PROGRAM C05_MachineStatus
VAR
	fbMachinState					: FB_SYSTEM_MachineState;

	fbPowerDelay					: TOF;
	tofEUCAPassthroughDisableDelay	: TOF;
	ftrigPassthroughCheck			: F_TRIG;
	ftrigConditionalRunOff			: F_TRIG;

	tonPowerUpTimer				: TON;
	tonEUCAMachineRun			: TON;

END_VAR
VAR // added by the converter: edge detectors and wires of the graphical bodies
    _w1, _w2 : BOOL;
END_VAR

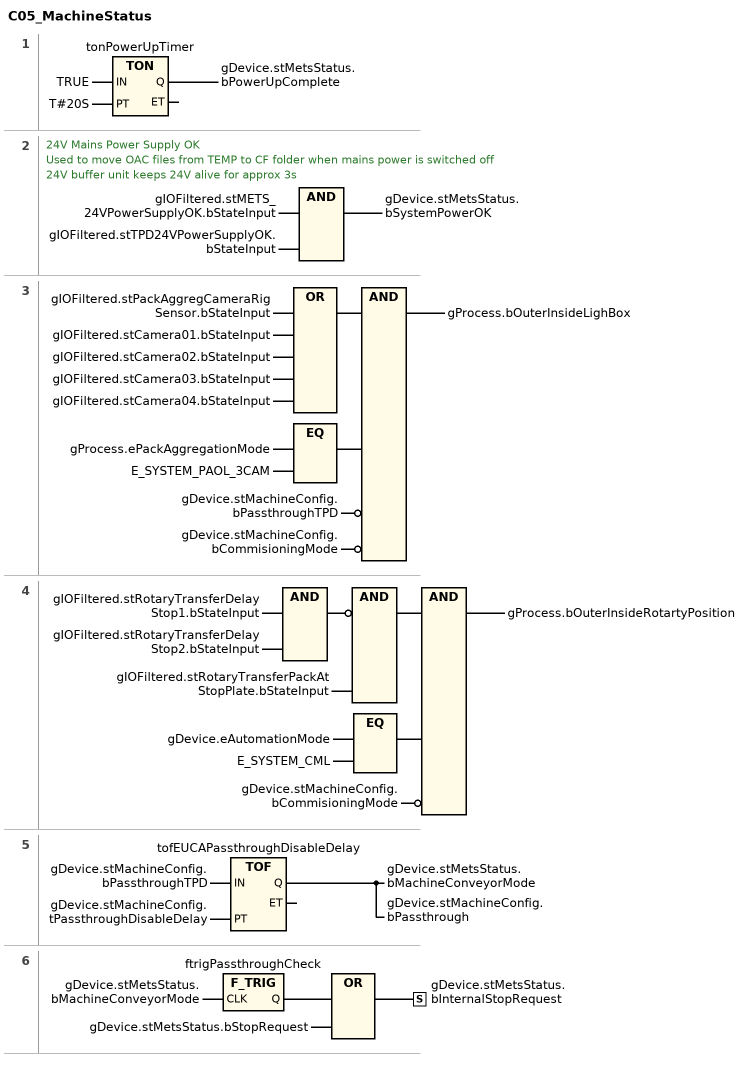
// NETWORK 1
tonPowerUpTimer(IN := TRUE, PT := T#20S); // TON
gDevice.stMetsStatus.bPowerUpComplete := tonPowerUpTimer.Q;

// NETWORK 2
// 					24V Mains Power Supply OK
// Used to move OAC files from TEMP to CF folder when mains power is switched off
// 24V buffer unit keeps 24V alive for approx 3s
//
gDevice.stMetsStatus.bSystemPowerOK := gIOFiltered.stMETS_24VPowerSupplyOK.bStateInput AND gIOFiltered.stTPD24VPowerSupplyOK.bStateInput;

// NETWORK 3
gProcess.bOuterInsideLighBox := (gIOFiltered.stPackAggregCameraRigSensor.bStateInput OR gIOFiltered.stCamera01.bStateInput OR gIOFiltered.stCamera02.bStateInput OR gIOFiltered.stCamera03.bStateInput OR gIOFiltered.stCamera04.bStateInput) AND gProcess.ePackAggregationMode = E_SYSTEM_PAOL_3CAM AND NOT gDevice.stMachineConfig.bPassthroughTPD AND NOT gDevice.stMachineConfig.bCommisioningMode;

// NETWORK 4
gProcess.bOuterInsideRotartyPosition := (NOT (gIOFiltered.stRotaryTransferDelayStop1.bStateInput AND gIOFiltered.stRotaryTransferDelayStop2.bStateInput) AND gIOFiltered.stRotaryTransferPackAtStopPlate.bStateInput) AND gDevice.eAutomationMode = E_SYSTEM_CML AND NOT gDevice.stMachineConfig.bCommisioningMode;

// NETWORK 5
tofEUCAPassthroughDisableDelay(IN := gDevice.stMachineConfig.bPassthroughTPD, PT := gDevice.stMachineConfig.tPassthroughDisableDelay); // TOF
gDevice.stMetsStatus.bMachineConveyorMode := tofEUCAPassthroughDisableDelay.Q;
gDevice.stMachineConfig.bPassthrough := tofEUCAPassthroughDisableDelay.Q;

// NETWORK 6
ftrigPassthroughCheck(CLK := gDevice.stMetsStatus.bMachineConveyorMode); // F_TRIG
gDevice.stMetsStatus.bInternalStopRequest S= ftrigPassthroughCheck.Q OR gDevice.stMetsStatus.bStopRequest;

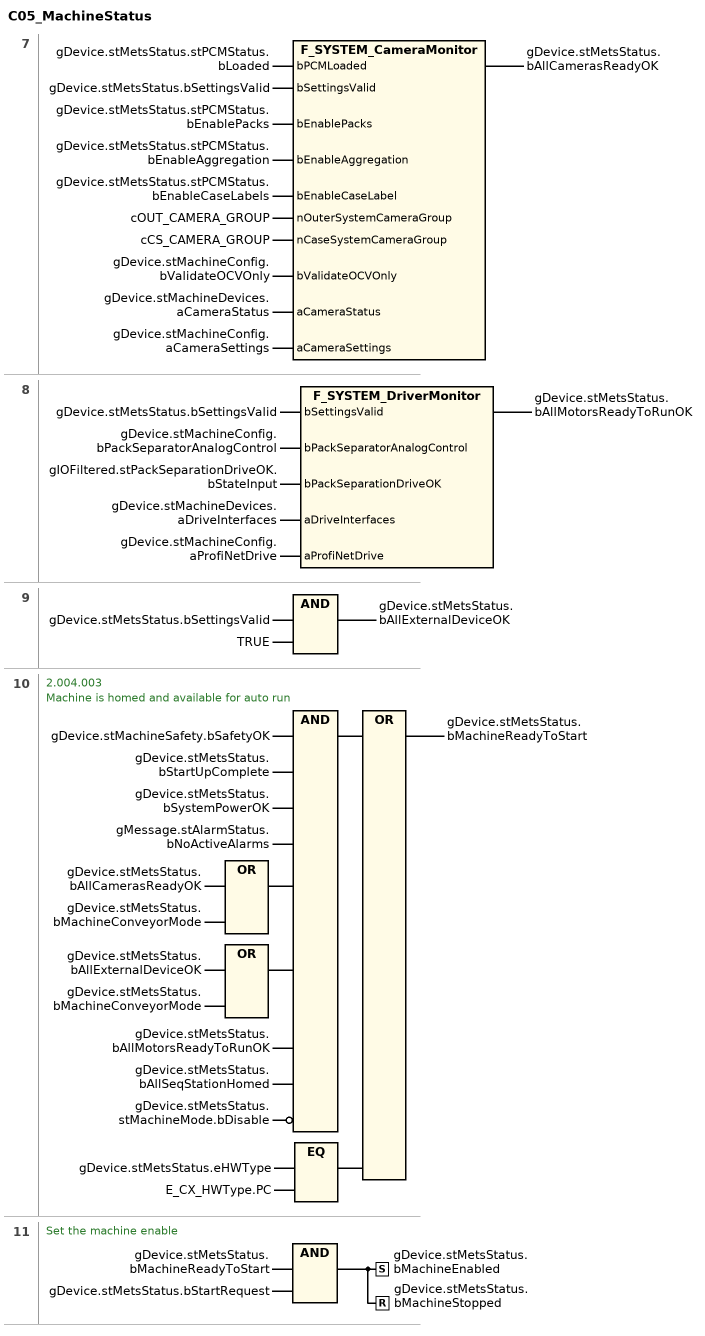
// NETWORK 7
gDevice.stMetsStatus.bAllCamerasReadyOK := F_SYSTEM_CameraMonitor(bPCMLoaded := gDevice.stMetsStatus.stPCMStatus.bLoaded, bSettingsValid := gDevice.stMetsStatus.bSettingsValid, bEnablePacks := gDevice.stMetsStatus.stPCMStatus.bEnablePacks, bEnableAggregation := gDevice.stMetsStatus.stPCMStatus.bEnableAggregation, bEnableCaseLabel := gDevice.stMetsStatus.stPCMStatus.bEnableCaseLabels, nOuterSystemCameraGroup := cOUT_CAMERA_GROUP, nCaseSystemCameraGroup := cCS_CAMERA_GROUP, bValidateOCVOnly := gDevice.stMachineConfig.bValidateOCVOnly, aCameraStatus := gDevice.stMachineDevices.aCameraStatus, aCameraSettings := gDevice.stMachineConfig.aCameraSettings);

// NETWORK 8
gDevice.stMetsStatus.bAllMotorsReadyToRunOK := F_SYSTEM_DriverMonitor(bSettingsValid := gDevice.stMetsStatus.bSettingsValid, bPackSeparatorAnalogControl := gDevice.stMachineConfig.bPackSeparatorAnalogControl, bPackSeparationDriveOK := gIOFiltered.stPackSeparationDriveOK.bStateInput, aDriveInterfaces := gDevice.stMachineDevices.aDriveInterfaces, aProfiNetDrive := gDevice.stMachineConfig.aProfiNetDrive);

// NETWORK 9
gDevice.stMetsStatus.bAllExternalDeviceOK := gDevice.stMetsStatus.bSettingsValid AND TRUE;

// NETWORK 10
// 					2.004.003
// Machine is homed and available for auto run
//
gDevice.stMetsStatus.bMachineReadyToStart := gDevice.stMachineSafety.bSafetyOK AND gDevice.stMetsStatus.bStartUpComplete AND gDevice.stMetsStatus.bSystemPowerOK AND gMessage.stAlarmStatus.bNoActiveAlarms AND (gDevice.stMetsStatus.bAllCamerasReadyOK OR gDevice.stMetsStatus.bMachineConveyorMode) AND (gDevice.stMetsStatus.bAllExternalDeviceOK OR gDevice.stMetsStatus.bMachineConveyorMode) AND gDevice.stMetsStatus.bAllMotorsReadyToRunOK AND gDevice.stMetsStatus.bAllSeqStationHomed AND NOT gDevice.stMetsStatus.stMachineMode.bDisable OR gDevice.stMetsStatus.eHWType = E_CX_HWType.PC;

// NETWORK 11
// Set the machine enable
_w1 := gDevice.stMetsStatus.bMachineReadyToStart AND gDevice.stMetsStatus.bStartRequest;
gDevice.stMetsStatus.bMachineEnabled S= _w1;
gDevice.stMetsStatus.bMachineStopped R= _w1;

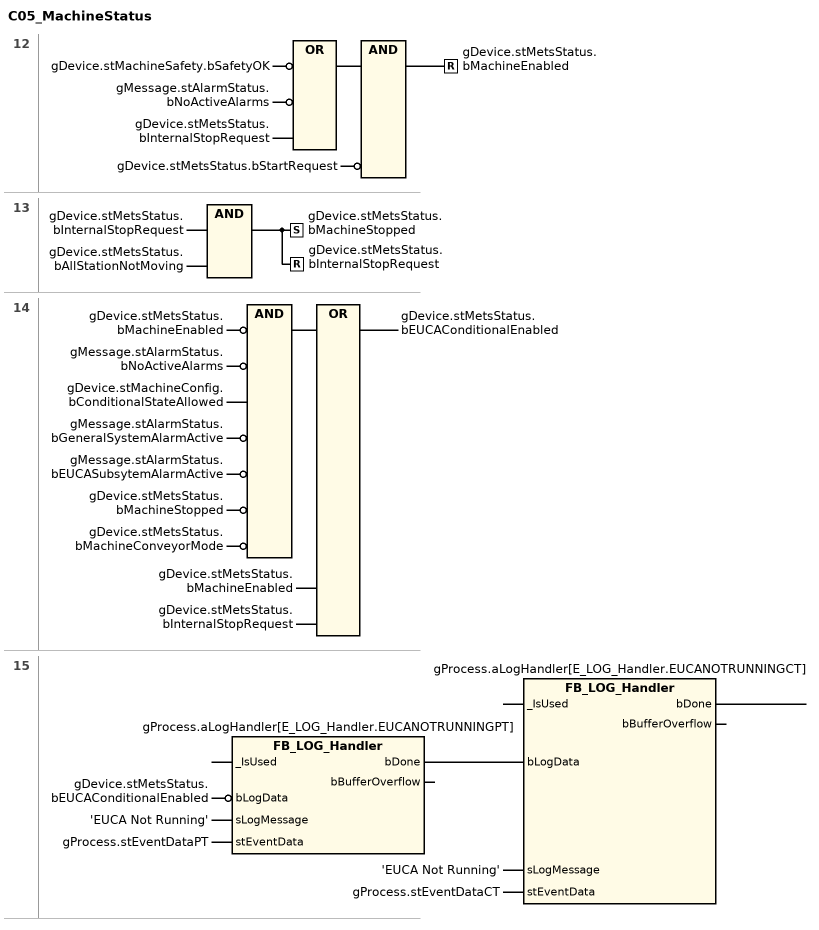
// NETWORK 12
gDevice.stMetsStatus.bMachineEnabled R= (NOT gDevice.stMachineSafety.bSafetyOK OR NOT gMessage.stAlarmStatus.bNoActiveAlarms OR gDevice.stMetsStatus.bInternalStopRequest) AND NOT gDevice.stMetsStatus.bStartRequest;

// NETWORK 13
_w2 := gDevice.stMetsStatus.bInternalStopRequest AND gDevice.stMetsStatus.bAllStationNotMoving;
gDevice.stMetsStatus.bMachineStopped S= _w2;
gDevice.stMetsStatus.bInternalStopRequest R= _w2;

// NETWORK 14
gDevice.stMetsStatus.bEUCAConditionalEnabled := NOT gDevice.stMetsStatus.bMachineEnabled AND NOT gMessage.stAlarmStatus.bNoActiveAlarms AND gDevice.stMachineConfig.bConditionalStateAllowed AND NOT gMessage.stAlarmStatus.bGeneralSystemAlarmActive AND NOT gMessage.stAlarmStatus.bEUCASubsytemAlarmActive AND NOT gDevice.stMetsStatus.bMachineStopped AND NOT gDevice.stMetsStatus.bMachineConveyorMode OR gDevice.stMetsStatus.bMachineEnabled OR gDevice.stMetsStatus.bInternalStopRequest;

// NETWORK 15
gProcess.aLogHandler[E_LOG_Handler.EUCANOTRUNNINGPT](
    bLogData := NOT gDevice.stMetsStatus.bEUCAConditionalEnabled,
    sLogMessage := 'EUCA Not Running',
    stEventData := gProcess.stEventDataPT); // FB_LOG_Handler
gProcess.aLogHandler[E_LOG_Handler.EUCANOTRUNNINGCT](
    bLogData := gProcess.aLogHandler[E_LOG_Handler.EUCANOTRUNNINGPT].bDone,
    sLogMessage := 'EUCA Not Running',
    stEventData := gProcess.stEventDataCT); // FB_LOG_Handler

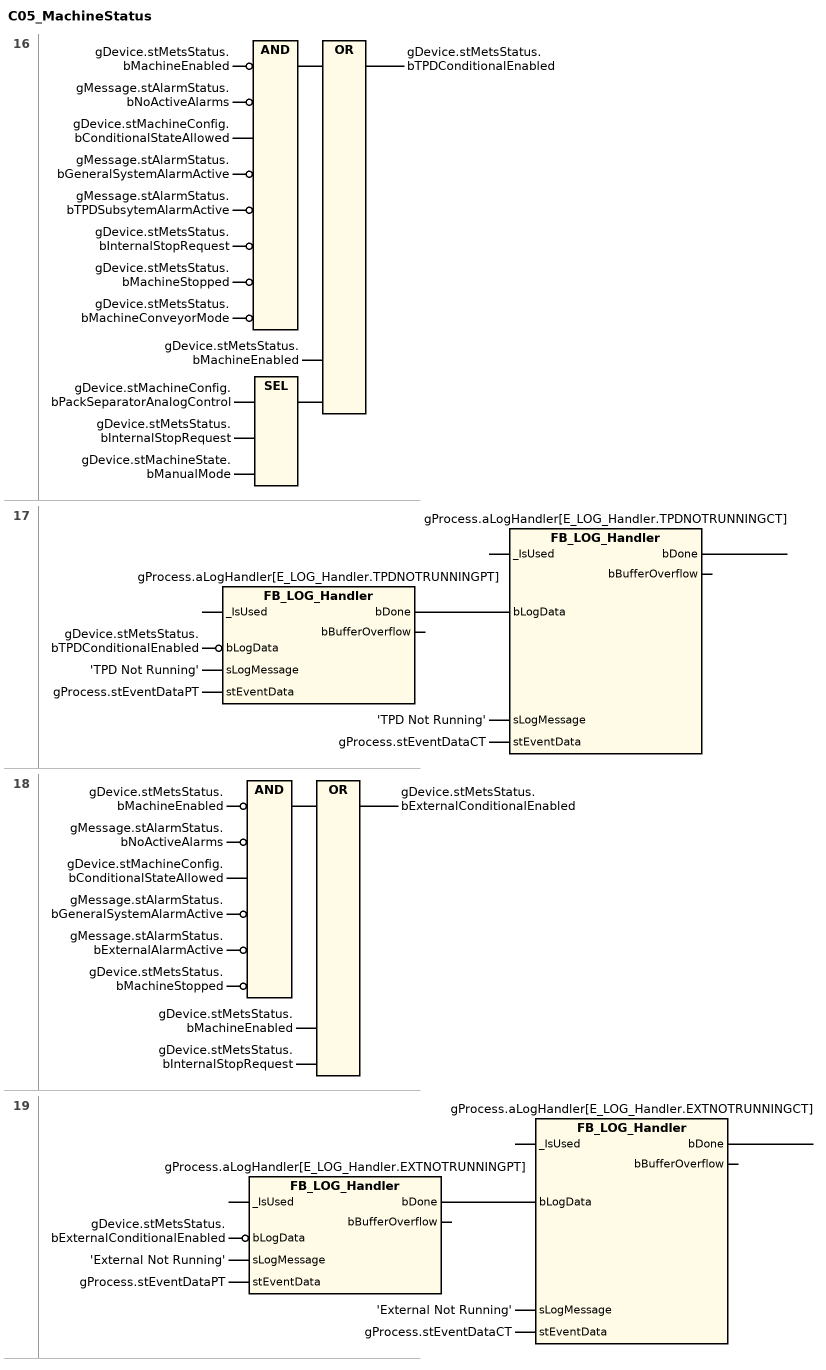
// NETWORK 16
gDevice.stMetsStatus.bTPDConditionalEnabled := NOT gDevice.stMetsStatus.bMachineEnabled AND NOT gMessage.stAlarmStatus.bNoActiveAlarms AND gDevice.stMachineConfig.bConditionalStateAllowed AND NOT gMessage.stAlarmStatus.bGeneralSystemAlarmActive AND NOT gMessage.stAlarmStatus.bTPDSubsytemAlarmActive AND NOT gDevice.stMetsStatus.bInternalStopRequest AND NOT gDevice.stMetsStatus.bMachineStopped AND NOT gDevice.stMetsStatus.bMachineConveyorMode OR gDevice.stMetsStatus.bMachineEnabled OR SEL(gDevice.stMachineConfig.bPackSeparatorAnalogControl, gDevice.stMetsStatus.bInternalStopRequest, gDevice.stMachineState.bManualMode);

// NETWORK 17
gProcess.aLogHandler[E_LOG_Handler.TPDNOTRUNNINGPT](
    bLogData := NOT gDevice.stMetsStatus.bTPDConditionalEnabled,
    sLogMessage := 'TPD Not Running',
    stEventData := gProcess.stEventDataPT); // FB_LOG_Handler
gProcess.aLogHandler[E_LOG_Handler.TPDNOTRUNNINGCT](
    bLogData := gProcess.aLogHandler[E_LOG_Handler.TPDNOTRUNNINGPT].bDone,
    sLogMessage := 'TPD Not Running',
    stEventData := gProcess.stEventDataCT); // FB_LOG_Handler

// NETWORK 18
gDevice.stMetsStatus.bExternalConditionalEnabled := NOT gDevice.stMetsStatus.bMachineEnabled AND NOT gMessage.stAlarmStatus.bNoActiveAlarms AND gDevice.stMachineConfig.bConditionalStateAllowed AND NOT gMessage.stAlarmStatus.bGeneralSystemAlarmActive AND NOT gMessage.stAlarmStatus.bExternalAlarmActive AND NOT gDevice.stMetsStatus.bMachineStopped OR gDevice.stMetsStatus.bMachineEnabled OR gDevice.stMetsStatus.bInternalStopRequest;

// NETWORK 19
gProcess.aLogHandler[E_LOG_Handler.EXTNOTRUNNINGPT](
    bLogData := NOT gDevice.stMetsStatus.bExternalConditionalEnabled,
    sLogMessage := 'External Not Running',
    stEventData := gProcess.stEventDataPT); // FB_LOG_Handler
gProcess.aLogHandler[E_LOG_Handler.EXTNOTRUNNINGCT](
    bLogData := gProcess.aLogHandler[E_LOG_Handler.EXTNOTRUNNINGPT].bDone,
    sLogMessage := 'External Not Running',
    stEventData := gProcess.stEventDataCT); // FB_LOG_Handler

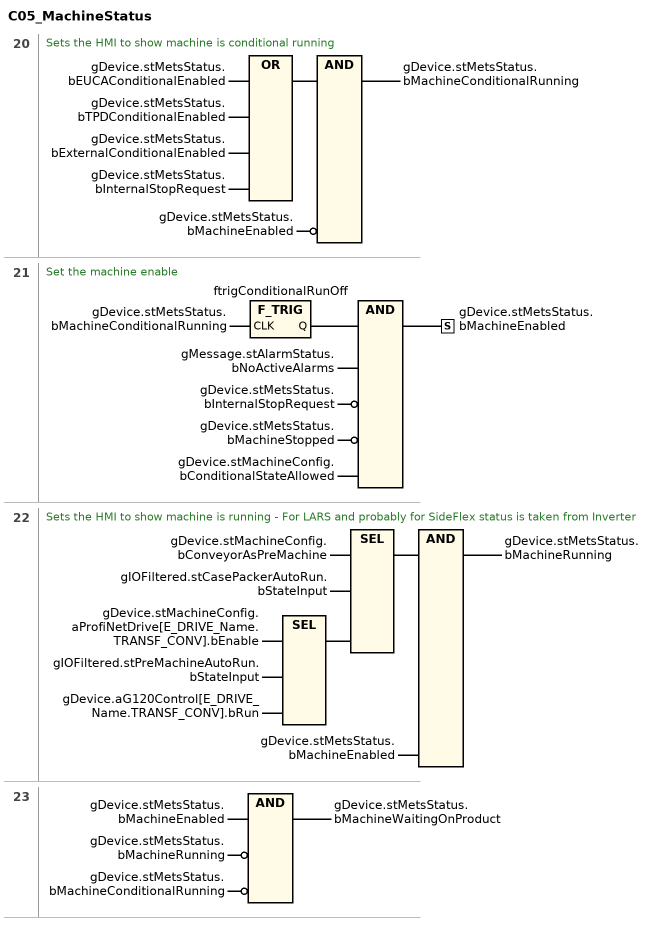
// NETWORK 20
// Sets the HMI to show machine is conditional running
gDevice.stMetsStatus.bMachineConditionalRunning := (gDevice.stMetsStatus.bEUCAConditionalEnabled OR gDevice.stMetsStatus.bTPDConditionalEnabled OR gDevice.stMetsStatus.bExternalConditionalEnabled OR gDevice.stMetsStatus.bInternalStopRequest) AND NOT gDevice.stMetsStatus.bMachineEnabled;

// NETWORK 21
// Set the machine enable
ftrigConditionalRunOff(CLK := gDevice.stMetsStatus.bMachineConditionalRunning); // F_TRIG
gDevice.stMetsStatus.bMachineEnabled S= ftrigConditionalRunOff.Q AND gMessage.stAlarmStatus.bNoActiveAlarms AND NOT gDevice.stMetsStatus.bInternalStopRequest AND NOT gDevice.stMetsStatus.bMachineStopped AND gDevice.stMachineConfig.bConditionalStateAllowed;

// NETWORK 22
// Sets the HMI to show machine is running - For LARS and probably for SideFlex status is taken from Inverter
gDevice.stMetsStatus.bMachineRunning := SEL(gDevice.stMachineConfig.bConveyorAsPreMachine, gIOFiltered.stCasePackerAutoRun.bStateInput, SEL(gDevice.stMachineConfig.aProfiNetDrive[E_DRIVE_Name.TRANSF_CONV].bEnable, gIOFiltered.stPreMachineAutoRun.bStateInput, gDevice.aG120Control[E_DRIVE_Name.TRANSF_CONV].bRun)) AND gDevice.stMetsStatus.bMachineEnabled;

// NETWORK 23
gDevice.stMetsStatus.bMachineWaitingOnProduct := gDevice.stMetsStatus.bMachineEnabled AND NOT gDevice.stMetsStatus.bMachineRunning AND NOT gDevice.stMetsStatus.bMachineConditionalRunning;

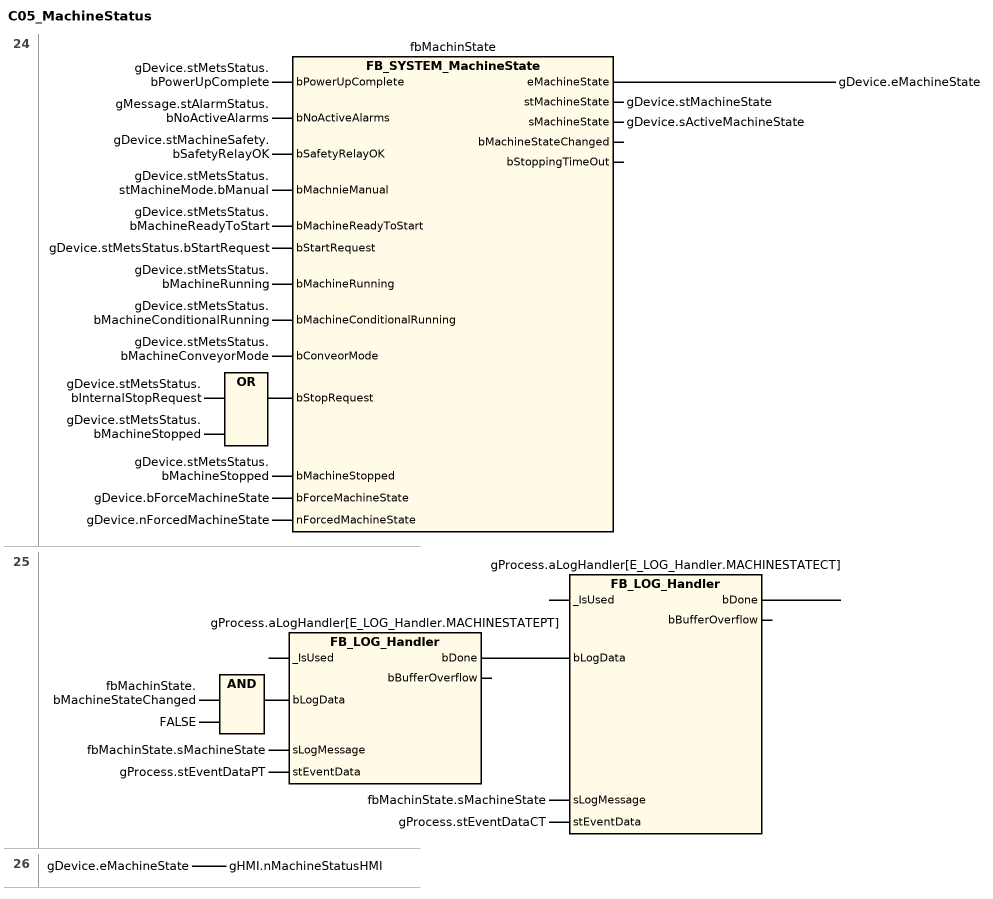
// NETWORK 24
fbMachinState(
    bPowerUpComplete := gDevice.stMetsStatus.bPowerUpComplete,
    bNoActiveAlarms := gMessage.stAlarmStatus.bNoActiveAlarms,
    bSafetyRelayOK := gDevice.stMachineSafety.bSafetyRelayOK,
    bMachnieManual := gDevice.stMetsStatus.stMachineMode.bManual,
    bMachineReadyToStart := gDevice.stMetsStatus.bMachineReadyToStart,
    bStartRequest := gDevice.stMetsStatus.bStartRequest,
    bMachineRunning := gDevice.stMetsStatus.bMachineRunning,
    bMachineConditionalRunning := gDevice.stMetsStatus.bMachineConditionalRunning,
    bConveorMode := gDevice.stMetsStatus.bMachineConveyorMode,
    bStopRequest := gDevice.stMetsStatus.bInternalStopRequest OR gDevice.stMetsStatus.bMachineStopped,
    bMachineStopped := gDevice.stMetsStatus.bMachineStopped,
    bForceMachineState := gDevice.bForceMachineState,
    nForcedMachineState := gDevice.nForcedMachineState,
    stMachineState => gDevice.stMachineState,
    sMachineState => gDevice.sActiveMachineState); // FB_SYSTEM_MachineState
gDevice.eMachineState := fbMachinState.eMachineState;

// NETWORK 25
gProcess.aLogHandler[E_LOG_Handler.MACHINESTATEPT](
    bLogData := fbMachinState.bMachineStateChanged AND FALSE,
    sLogMessage := fbMachinState.sMachineState,
    stEventData := gProcess.stEventDataPT); // FB_LOG_Handler
gProcess.aLogHandler[E_LOG_Handler.MACHINESTATECT](
    bLogData := gProcess.aLogHandler[E_LOG_Handler.MACHINESTATEPT].bDone,
    sLogMessage := fbMachinState.sMachineState,
    stEventData := gProcess.stEventDataCT); // FB_LOG_Handler

// NETWORK 26
gHMI.nMachineStatusHMI := gDevice.eMachineState;

END_PROGRAM

(* stored: Version 1.1.0.1
   POU C05_MachineStatus: Id {bd01ada0-da10-4b5a-93f5-f3c587c8bb54}, SpecialFunc None *)
